VAR_GLOBAL CONSTANT
	/// Reduced, was 300
	cintMaxDecisions: INT := 100;
END_VAR

(* stored: Version 1.1.0.1, ProductVersion 3.1.0.23
   GVL Const_DPJ: Id {f4f7fcb7-3d4c-4b0d-9783-33f888966e82} *)
